(* PLC project Basic FBD logic, react-plc-diagram PLCopen XML test fixtures 0.1.0 *)
(* stored: creationDateTime 2026-08-12T00:00:00Z, modificationDateTime 2026-08-12T00:00:00Z *)

PROGRAM BasicLogic
  VAR
    Start : BOOL;
    Safe : BOOL;
    Motor : BOOL;
  END_VAR

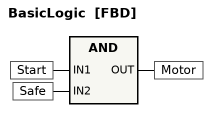
(* FBD diagram, written out as Structured Text *)
Motor := Start AND Safe;
END_PROGRAM
